{attribute 'linkalways'} 
{attribute 'no_explicit_call' := 'This FB is a CLASS and must be accessed using methods or properties'}
{attribute 'enable_dynamic_creation'}
FUNCTION_BLOCK FINAL LT_DINT EXTENDS Node
VAR
	in1 : _DINT(0);
	in2 : _DINT(0);
	out : _BOOL(FALSE);
END_VAR

METHOD PUBLIC Clone : I_Node
VAR
	pNode : POINTER TO LT_DINT;
END_VAR
pNode := __NEW(LT_DINT);
Clone := pNode^;
END_METHOD

METHOD FB_init : BOOL
VAR_INPUT
	bInitRetains : BOOL; // if TRUE, the retain variables are initialized (warm start / cold start)
	bInCopyCode : BOOL;  // if TRUE, the instance afterwards gets moved into the copy code (online change)
END_VAR
AddInput('in1',THIS^.in1);
AddInput('in2',THIS^.in2);
AddOutput('out', THIS^.out);
END_METHOD

METHOD PROTECTED OnExecute
VAR
END_VAR
out.Value := in1.Value < in2.Value;
END_METHOD

END_FUNCTION_BLOCK

(* stored: Version 1.1.0.1, ProductVersion 3.1.4024.15
   POU LT_DINT: Id {453f4ac4-866a-45e2-8a2f-de9834c2d980}, SpecialFunc None
   Folder Constructor: Id {b8b99cff-a060-4aa8-a544-51d4e639728a}
   Method Clone: Id {5edb6c7f-2a49-43c8-a828-0910883c2a99}
   Method FB_init: Id {f4e49e76-052a-485d-827a-d16f90d1ecd3}
   Method OnExecute: Id {fd5b1561-b717-412b-8d58-316955bc9085} *)
